Staubli VAL3: Form_PanelStr.pgx

public program Form_PanelStr(string x_sTitle, string x_sPanelTitle, string& x_sList[], bool& x_bList[], num& x_nSelectIndex, string x_sBottom)
  local num l_nNum
begin

//×××××××××××××××××××××××××××××××××××××××××××××××××
//×××××××××××××××××××××××××××××××××××××××××××××××××
if size(x_bList)!=size(x_sList)
  return
endIf
resize(sBuff,1,size(x_bList))

for l_nNum=0 to size(x_bList)-1
  if x_bList[l_nNum]
    sBuff[l_nNum]=toString("",l_nNum+1)+"."+"Pallet:"+x_sList[l_nNum]
  else
    sBuff[l_nNum]=toString("",l_nNum+1)+"."+"Point"
  endIf
endFor
//*********************************************************
call Form_PanelList(x_sTitle,x_sPanelTitle,sBuff,x_nSelectIndex,x_sBottom)



end
